// TIA Portal V16 export
// export: Created 2023-03-29T11:03:46.0979012Z, ExportSetting WithDefaults, DisplayName Totally Integrated Automation Portal, DisplayVersion V16 Update 6, DisplayName TIA Portal Version Control Interface, DisplayVersion V16 Update 2, DisplayName TIA Portal Openness, DisplayVersion V16 Update 6, DisplayName STEP 7 Professional, DisplayVersion V16 Update 6, DisplayName STEP 7 Safety, DisplayVersion V16, DisplayName WinCC Advanced, DisplayVersion V16 Update 6
VAR_GLOBAL   // PLC tag table "Analogi"
   AI_poziom_zbiornik_4 AT %MW42 : Word;
   AI_poziom_zbiornik_2 AT %MW38 : Word;
   IW68 AT %IW68 : Word;   // wejscie AI
   AI_poziom_zbiornik_1 AT %MW36 : Word;
   AI_poziom_zbiornik_3 AT %MW40 : Word;
   IW78 AT %IW78 : Word;   // wejscie AI
   AI_położenie_Z10 AT %MW34 : Word;
   AI_przepływ AT %MW30 : Word;
   AI_ciśnienie_B5 AT %MW32 : Word;
   IW70 AT %IW70 : Word;   // wejscie AI
   IW72 AT %IW72 : Word;   // wejscie AI
   IW76 AT %IW76 : Word;   // wejscie AI
   IW74 AT %IW74 : Word;   // wejscie AI
   switch_Kolman AT %M46.0 : Bool;   // przełącznik funkcji filtr analogów (Kolman = OFF, bez Kolman = ON)
   I AT %MW48 : Int;   // kalman zmienna przechwuje adres wejścia AI
END_VAR
